// SIMATIC S7-200 project (STEP 7-Micro/WIN), CPU 224 UN REL 02.02

ORGANIZATION_BLOCK MAIN:OB1
TITLE=PROGRAM COMMENTS
BEGIN
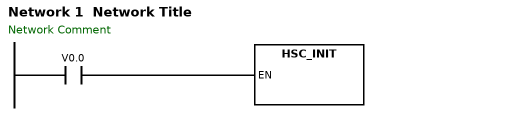
Network 1 // Network Title
// Network Comment
// (network saved uncompiled; LAD cells follow)
// row 0: c0 -| |- V0.0  c1 --  c2 [HSC_INIT EN:=power@row0]
END_ORGANIZATION_BLOCK

SUBROUTINE_BLOCK HSC_INIT:SBR1
TITLE=
BEGIN
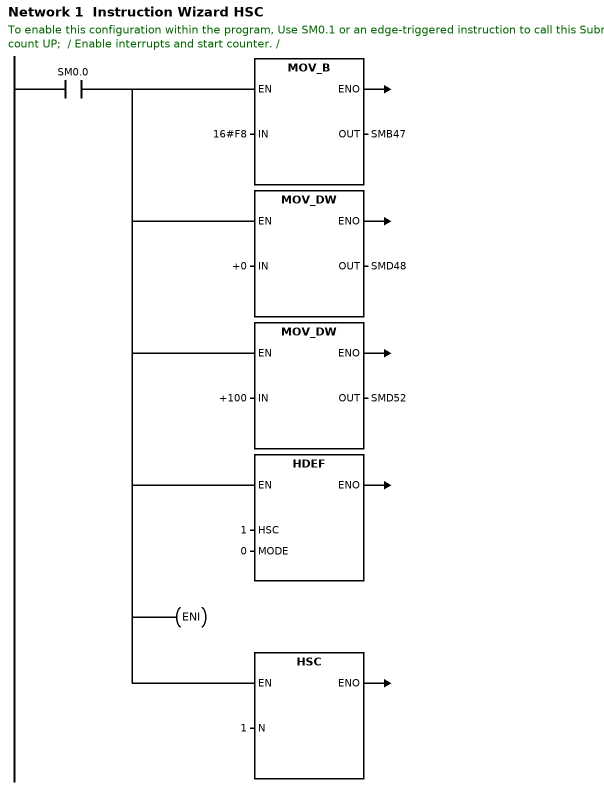
Network 1 // Instruction Wizard HSC
// To enable this configuration within the program, Use SM0.1 or an edge-triggered instruction to call this Subroutine once from the MAIN program block.  
// Configure HC1 for Mode 0; CV = 0; PV = 100; count UP; 
// Enable interrupts and start counter.
// 
//Set control bits: count UP; enabled; 
//Load CV
//Load PV
LD     SM0.0
MOVB   16#F8, SMB47
MOVD   +0, SMD48
MOVD   +100, SMD52
HDEF   1, 0
ENI
HSC    1
END_SUBROUTINE_BLOCK
